(* IEC 61131-3 sources: ia2/examples/device_health/pous, 1 file *)

(* ---- main.st ---- *)
PROGRAM main
VAR
    input_value : INT;
    ticks : DINT;
END_VAR
ticks := ticks + 1;
END_PROGRAM
